ABB RobotStudio station: Solution1_1_20220418-143055.rsstn

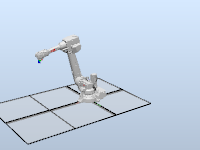
Station Solution1 (saved by RobotStudio 21.4.9700.0)
Controller IRB2600_12_185
  mechanical unit ROB_1: IRB2600_12_185__02, 6 joints, base frame (0, 0, 0) mm
Layout (positions relative to the parent item):
  - IRB2600_12_185__02 [mechanism, from Robots\IRB2600_12_185_G_02.rslib] at (0, 0, 0) mm; joint values [0.0004, 0.2608, -0.0544, -0.0092, 1.3475, -0.0032] (rad or m)
